(* CoDeSys 2.3 export: FGETK14PUMP.EXP *)

(* POU K14/fGetK14Pump, ST *)
FUNCTION fGetK14Pump :BOOL
(* Проверка включения насоса*)
VAR_INPUT
	PumpID : USINT;
END_VAR
fGetK14Pump := MU110DO.K14PumpIsOn[PumpID];
END_FUNCTION
